(* PLC project OOP_Curso, Beckhoff Automation GmbH TwinCAT PLC Control 3.5.13.21 *)
(* stored: creationDateTime 2023-09-16T13:26:48.8044251, modificationDateTime 2023-09-16T13:26:48.8083286 *)

INTERFACE I_AveCorredora
METHOD Correr : BOOL
END_METHOD
END_INTERFACE

INTERFACE I_AveNadadora
METHOD Nadar : BOOL
END_METHOD
END_INTERFACE

INTERFACE I_AveVoladora
METHOD Volar : BOOL
END_METHOD
END_INTERFACE

FUNCTION_BLOCK Aguila IMPLEMENTS I_AveVoladora
VAR_INPUT
    velocidad : REAL;
    alturaMaxima : REAL;
END_VAR
VAR
END_VAR

            
          

METHOD Volar : BOOL
                  Volar:= TRUE;
                
END_METHOD
END_FUNCTION_BLOCK

FUNCTION_BLOCK Avestruz IMPLEMENTS I_AveCorredora
VAR_INPUT
    velocidad : REAL;
    tiempoCorriendo : TIME;
END_VAR
VAR
END_VAR

            
          

METHOD Correr : BOOL
                  Correr := TRUE;
                
END_METHOD
END_FUNCTION_BLOCK

FUNCTION_BLOCK Pato IMPLEMENTS I_AveVoladora, I_AveNadadora
VAR_INPUT
    velocidad : REAL;
    alturaMaxima : REAL;
    tiempoBuceo : TIME;
END_VAR
VAR
END_VAR

            
          

METHOD Volar : BOOL
                  Volar := true;
                
END_METHOD

METHOD Nadar : BOOL
                  Nadar := TRUE;
                
END_METHOD
END_FUNCTION_BLOCK

PROGRAM _27_SOLID_ISP
VAR
	Patito_feo : Pato;
	Aguila_imperial : Aguila;
	Avestruz_de_cuello_azul : Avestruz;
END_VAR

            Patito_feo.Nadar();
Patito_feo.Volar();

Aguila_imperial.Volar();

Avestruz_de_cuello_azul.Correr();

          
END_PROGRAM
